// Boundaries indicating leak monitor locations
TYPE ST_LeakBoundaries :
STRUCT
	{attribute 'pytmc' := '
		pv: L_MIN01
		io: io
	'}
	nLMin1 : UINT;
	{attribute 'pytmc' := '
		pv: L_MAX01
		io: io
	'}
	nLMax1 : UINT;
	{attribute 'pytmc' := '
		pv: L_MIN02
		io: io
	'}
	nLMin2 : UINT;
	{attribute 'pytmc' := '
		pv: L_MAX02
		io: io
	'}
	nLMax2 : UINT;
	{attribute 'pytmc' := '
		pv: L_MIN03
		io: io
	'}
	nLMin3 : UINT;
	{attribute 'pytmc' := '
		pv: L_MAX03
		io: io
	'}
	nLMax3 : UINT;
	{attribute 'pytmc' := '
		pv: L_MIN04
		io: io
	'}
	nLMin4 : UINT;
	{attribute 'pytmc' := '
		pv: L_MAX04
		io: io
	'}
	nLMax4 : UINT;
	{attribute 'pytmc' := '
		pv: L_MIN05
		io: io
	'}
	nLMin5 : UINT;
	{attribute 'pytmc' := '
		pv: L_MAX05
		io: io
	'}
	nLMax5 : UINT;
	{attribute 'pytmc' := '
		pv: L_MIN06
		io: io
	'}
	nLMin6 : UINT;
	{attribute 'pytmc' := '
		pv: L_MAX06
		io: io
	'}
	nLMax6 : UINT;
END_STRUCT
END_TYPE

(* stored: Version 1.1.0.1, ProductVersion 3.1.4024.0
   DUT ST_LeakBoundaries: Id {984a6730-ff5d-4e76-ab98-a071061d040f} *)
